// TIA Portal V15.1 export
// export: Created 2020-06-12T07:35:38.3037109Z, ExportSetting None, DisplayName Totally Integrated Automation Portal, DisplayVersion V15.1, DisplayName TIA Portal Openness, DisplayVersion V15.1, DisplayName STEP 7 Professional, DisplayVersion V15.1, DisplayName STEP 7 Safety, DisplayVersion V15.1, DisplayName WinCC Advanced, DisplayVersion V15.1
DATA_BLOCK "Safety"   // DB608
{ S7_Optimized_Access := 'FALSE' }
   VAR
      ES1GD01_S34_on { ExternalWritable := 'False'} : Bool := TRUE;   // ES1GD01 Control Voltage ON
      ES1GD01_S43_off { ExternalWritable := 'False'} : Bool := FALSE;   // ES1GD01 Circuit Breaker off
      ES1GD01_S43_auto { ExternalWritable := 'False'} : Bool := TRUE;   // ES1GD01 Circuit Breaker auto
      ES1GD01_S48_rc_key { ExternalWritable := 'False'} : Bool := FALSE;   // ES1GD01 Remote Control Key
      ES1GD01_noemst { ExternalWritable := 'False'} : Bool := TRUE;   // Emergency Stop ES1GD01 ok
      ES1GD02_act { ExternalWritable := 'False'} : Bool := FALSE;   // Remote Control active
      ES1GD03_noemst { ExternalWritable := 'False'} : Bool := TRUE;   // Emergency Stop ES1GD03 ok
      ES1GT71_noemst { ExternalWritable := 'False'} : Bool := TRUE;   // Emergency Stop ES1GT71 ok
      ES1GT72_noemst { ExternalWritable := 'False'} : Bool := TRUE;   // Emergency Stop ES1GT72 ok
      ES1GT74_noemst { ExternalWritable := 'False'} : Bool := TRUE;   // SPARE Emergency Stop ES1GT74 ok
      ES1GT07_noemst { ExternalWritable := 'False'} : Bool := TRUE;   // Emergency Stop Portal Desk
      ES1YD01_noemst { ExternalWritable := 'False'} : Bool := TRUE;   // Emergency Stop ES1YD01 ok
      ES1YM01_emst_res { ExternalWritable := 'False'} : Bool := FALSE;   // Emergency Stop Reset
      ES1LE1_GY02_cls { ExternalWritable := 'False'} : Bool := TRUE;   // Safety door Top Platform closed
      ES1LE1_GY04_ncls { ExternalWritable := 'False'} : Bool := TRUE;   // Spindle Break not Closed
      ES1LE3_GY01_pos { ExternalWritable := 'False'} : Bool := FALSE;   // Hood Fitted
      ES1LE3_GY03_nlck { ExternalWritable := 'False'} : Bool := TRUE;   // Hood not Locked
      ES1LE4_GY01_cls { ExternalWritable := 'False'} : Bool := TRUE;   // Ladder Hood closed
      ES1GT07_SP52 { ExternalWritable := 'False'} : Bool := FALSE;   // Hood upwards
      ES1GT07_SP57 { ExternalWritable := 'False'} : Bool := FALSE;   // Hood downwards
      ES1GD01_S43 { ExternalWritable := 'False'} : Bool := FALSE;   // Circuit Breaker switch Auto mode
      ES1LS1_XS01_GY01_cls { ExternalWritable := 'False'} : Bool := FALSE;
      ES1LT1_XS01_GY01_cls { ExternalWritable := 'False'} : Bool := FALSE;
      ___outputs___ { ExternalAccessible := 'False'; ExternalVisible := 'False'; ExternalWritable := 'False'} : Int := 0;
      emer_undel_on { ExternalWritable := 'False'} : Bool := TRUE;   // Emergency line Undelayed ok
      emer_del_on { ExternalWritable := 'False'} : Bool := TRUE;   // Emergency line Delayed ok
      sd_undel_on { ExternalWritable := 'False'} : Bool := TRUE;   // Emergency & SDoors line Undelayed ok
      sd_del_on { ExternalWritable := 'False'} : Bool := TRUE;   // Emergency & SDoors line Delayed ok
      mcb_rel_undel { ExternalWritable := 'False'} : Bool := FALSE;   // MCB release undelayed ok
      mcb_rel_del { ExternalWritable := 'False'} : Bool := FALSE;   // MCB release delayed ok
      ES1YM01_emer_undel_on { ExternalWritable := 'False'} : Bool := TRUE;   // Emergency line Undelayed out
      ES1YM01_emer_undel_err { ExternalWritable := 'False'} : Bool := FALSE;   // Emergency line Undelayed error
      ES1YM01_emer_del_on { ExternalWritable := 'False'} : Bool := TRUE;   // Emergency line Delayed out
      ES1YM01_emer_del_err { ExternalWritable := 'False'} : Bool := FALSE;   // Emergency line Delayed error
      ES1LA1_M01_rel_err { ExternalWritable := 'False'} : Bool := FALSE;   // Screw Conveyer release Error
      ES1LE1_EV02_rel_on { ExternalWritable := 'False'} : Bool := TRUE;   // Spindle Break Release on
      ES1LE1_EV02_rel_err { ExternalWritable := 'False'} : Bool := FALSE;   // Spindle Break Release error
      ES1LE1_M01_rel_on { ExternalWritable := 'False'} : Bool := TRUE;   // Electrode Carriage Safe Release on
      ES1LE1_M01_rel_err { ExternalWritable := 'False'} : Bool := FALSE;   // Electrode Carriage Safe Release error
      ES1LE2_M01_rel_err { ExternalWritable := 'False'} : Bool := FALSE;   // X-Drive Safe Release error
      ES1LE2_M02_rel_err { ExternalWritable := 'False'} : Bool := FALSE;   // Y-Drive Safe Release error
      ES1LE3_M01_rel_on { ExternalWritable := 'False'} : Bool := TRUE;   // Protective Gas Hood Safe Release on
      ES1LE3_M01_rel_err { ExternalWritable := 'False'} : Bool := FALSE;   // Protective Gas Hood Safe Release error
      ES1LE4_EV01_rel_on { ExternalWritable := 'False'} : Bool := TRUE;   // Pneumatic Valve Power Ram Safe Release on
      ES1LE4_EV01_rel_err { ExternalWritable := 'False'} : Bool := FALSE;   // Pneumatic Valve Power Ram Safe Release error
      ES1LE4_EV02_rel_on { ExternalWritable := 'False'} : Bool := TRUE;   // Pneumatic Valve Current Pipes Cylinders Safe Release on
      ES1LE4_EV02_rel_err { ExternalWritable := 'False'} : Bool := FALSE;   // Pneumatic Valve Current Pipes Cylinders Safe Release error
      ES1LE4_M01_rel_on { ExternalWritable := 'False'} : Bool := TRUE;   // Portal Swiveling Safe Release on
      ES1LE4_M01_rel_err { ExternalWritable := 'False'} : Bool := FALSE;   // Portal Swiveling Safe Release error
      ES1LM1_EV01_rel_on { ExternalWritable := 'False'} : Bool := TRUE;   // Pneumatic Valve Baseplate Clamp MS1 Cylinders Safe Release on
      ES1LM1_EV01_rel_err { ExternalWritable := 'False'} : Bool := FALSE;   // Pneumatic Valve Baseplate Clamp MS1 Cylinders Safe Release error
      ES1LM2_EV01_rel_on { ExternalWritable := 'False'} : Bool := TRUE;   // Pneumatic Valve Baseplate Clamp MS2 Cylinders Safe Release on
      ES1LM2_EV01_rel_err { ExternalWritable := 'False'} : Bool := FALSE;   // Pneumatic Valve Baseplate Clamp MS2 Cylinders Safe Release error
      ES1LS1_XS01_rel_on { ExternalWritable := 'False'} : Bool := TRUE;   // MCB Safety Release on
      ES1LS1_XS01_rel_err { ExternalWritable := 'False'} : Bool := FALSE;   // MCB Safety Release error
      ES1LE1_M01_STO { ExternalWritable := 'False'} : Bool := TRUE;   // Electrode Carriage Safe Torque off Ok
      ES1LE1_M01_STO_err { ExternalWritable := 'False'} : Bool := FALSE;   // Electrode Carriage Safe Torque off error
      ES1LE3_M01_STO { ExternalWritable := 'False'} : Bool := TRUE;   // Protective Gas Hood Safe Torque off Ok
      ES1LE3_M01_STO_err { ExternalWritable := 'False'} : Bool := FALSE;   // Protective Gas Hood Safe Torque off error
      ES1LE4_M01_STO { ExternalWritable := 'False'} : Bool := TRUE;   // Portal Swiveling Safe Torque off Ok
      ES1LE4_M01_STO_err { ExternalWritable := 'False'} : Bool := FALSE;   // Portal Swiveling Safe Torque off error
   END_VAR
BEGIN
END_DATA_BLOCK
